Yaskawa INFORM job: pipe_junction_cylinder_program.JBI

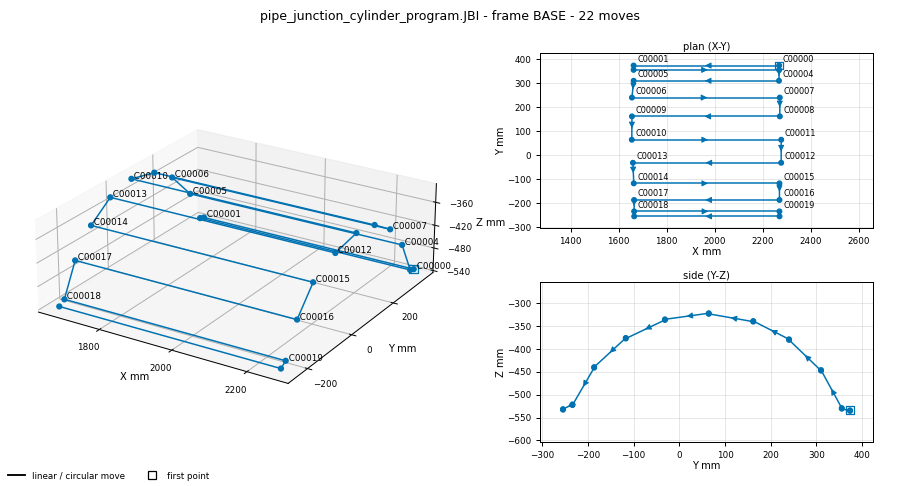
[picture p0: tool path of pipe_junction_cylinder_program.JBI in frame BASE, 22 of 25 moves have a stored position in this frame; points joined in program order, loops and branches not executed]
/JOB
//NAME pipe_junction_cylinder_program
//POS
///NPOS 22,0,22,0,0,0
///TOOL 0
///POSTYPE BASE
///RECTAN
///RCONF 0,0,0,0,0,0,0,0,0,0,0,0,0,0,0,0,0,0,0,0,0,0,0,0
C00000=2268.474795,373.539391,-534.065209,175.000000,-60.000000,-89.987700
C00001=1662.292449,373.539384,-535.404354,175.000000,-60.000000,-89.987700
C00002=1662.251200,355.445636,-530.584844,-175.000000,-70.069070,-89.954103
C00003=2268.337127,355.445642,-529.245912,-175.000000,-70.069070,-89.954103
C00004=2267.679681,310.079646,-445.993675,-175.000000,-52.757911,-89.903777
C00005=1662.477078,310.079640,-447.330656,-175.000000,-52.757911,-89.903777
C00006=1655.312989,240.061472,-379.997259,-175.000000,-35.016107,-89.819340
C00007=2270.993588,240.061479,-378.637131,-175.000000,-35.016107,-89.819340
C00008=2271.302511,161.742944,-338.737994,161.023875,-5.000000,5.000000
C00009=1655.411283,161.742938,-340.098587,161.023875,-5.000000,5.000000
C00010=1654.753651,64.450756,-323.023146,175.000000,-5.000000,5.000000
C00011=2276.975786,64.450763,-321.648567,175.000000,-5.000000,5.000000
C00012=2276.821776,-31.499366,-334.981563,-163.243910,-5.000000,-5.000000
C00013=1659.449481,-31.499373,-336.345428,-163.243910,-5.000000,-5.000000
C00014=1662.963205,-117.178446,-377.050687,175.000000,-34.076390,89.812884
C00015=2269.649089,-117.178439,-375.710430,175.000000,-34.076390,89.812884
C00016=2269.812232,-186.367272,-439.479303,175.000000,-51.255425,89.898433
C00017=1664.417008,-186.367279,-440.816709,175.000000,-51.255425,89.898433
C00018=1664.534822,-233.832301,-522.678117,-175.000000,-68.532601,89.950225
C00019=2269.584715,-233.832294,-521.341474,-175.000000,-68.532601,89.950225
C00020=2269.940432,-254.640841,-531.484739,175.000000,-60.000000,89.985692
C00021=1664.702128,-254.640848,-532.821798,175.000000,-60.000000,89.985692
///POSTYPE PULSE
///PULSE
EX00000=366592.0
///POSTYPE PULSE
///PULSE
EC00000=366592.0
EC00001=366592.0
EC00002=366592.0
EC00003=366592.0
EC00004=366592.0
EC00005=366592.0
EC00006=366592.0
EC00007=366592.0
EC00008=366592.0
EC00009=366592.0
EC00010=366592.0
EC00011=366592.0
EC00012=366592.0
EC00013=366592.0
EC00014=366592.0
EC00015=366592.0
EC00016=366592.0
EC00017=366592.0
EC00018=366592.0
EC00019=366592.0
EC00020=366592.0
EC00021=366592.0
//INST
///DATE 2023/08/15 17:09
///ATTR SC,RW,RJ
////FRAME BASE
///GROUP1 RB1,ST1
NOP
MOVJ P009 EX000 VJ=15.00
MOVJ C00000 EC00000 VJ=15.0
CALL JOB:SPYON
MOVL C00001 EC00001 V=150.0
MOVL C00002 EC00002 V=150.0
MOVL C00003 EC00003 V=150.0
MOVL C00004 EC00004 V=150.0
MOVL C00005 EC00005 V=150.0
MOVL C00006 EC00006 V=150.0
MOVL C00007 EC00007 V=150.0
MOVL C00008 EC00008 V=150.0
MOVL C00009 EC00009 V=150.0
MOVL C00010 EC00010 V=150.0
MOVL C00011 EC00011 V=150.0
MOVL C00012 EC00012 V=150.0
MOVL C00013 EC00013 V=150.0
MOVL C00014 EC00014 V=150.0
MOVL C00015 EC00015 V=150.0
MOVL C00016 EC00016 V=150.0
MOVL C00017 EC00017 V=150.0
MOVL C00018 EC00018 V=150.0
MOVL C00019 EC00019 V=150.0
MOVL C00020 EC00020 V=150.0
MOVL C00021 EC00021 V=150.0
CALL JOB:SPYOF
MOVJ P009 VJ=15.00
MOVL P009 EX00000 V=150.0
END
